FUNCTION_BLOCK FB_ManualMotionControl
VAR_INPUT
	
END_VAR
VAR_OUTPUT
END_VAR
VAR_IN_OUT
	stServoInterface		: stServoInterface;
END_VAR
VAR
	
	servoPower				: MC_Power;
	servoBuffer				: MC_BufferMode := MC_Aborting;
	
	servoReset				: MC_Reset;
	servoHome				: MC_Home;
	
	servoStatus				: MC_ReadStatus;
	
	servoSetPosition		: MC_SetPosition;
	
	servoJog				: MC_Jog;
	
	servoStop				: MC_Stop;
	
	servoMoveAbsolute		: MC_MoveAbsolute;
	
	servoMoveRelative		: MC_MoveRelative;
	
	servoMoveVelocity		: MC_MoveVelocity;
	
	jogErrorID				: UDINT;
	
	errorStop: BOOL;
	disabled: BOOL;
	stopping: BOOL;
	discreteMotion: BOOL;
	continuousMotion: BOOL;
	syncMotion: BOOL;
	homing: BOOL;
	constVelocity: BOOL;
	accel: BOOL;
	decel: BOOL;
	status: ST_AxisStatus;
	
	powerInterface 		: mcInterface;
	resetInterface		: mcInterface;
	homeInterface		: mcInterface;
	jogInterface		: mcInterface;
	stopInterface		: mcInterface;
	moveAbsInterface	: mcInterface;
	moveRelInterface	: mcInterface;
	moveVelInterface	: mcInterface;
	statusInterface		: mcInterface;
	
	// State Machine Variables
	startCycle			: BOOL;
	continueToTop		: BOOL;
	continueToBottom	: BOOL;
	endAtTop			: BOOL;
	endAtBottom			: BOOL;
	moveBottomTrig			: BOOL;
	moveTopTrig				: BOOL;
	
	demoState			: FB_ManualStateMachine;
	demoModePermissive	: BOOL;
	demoModeRun			: BOOL;
	bottomComplete		: BOOL;
	topComplete			: BOOL;
	
	servoMoveBottom		: MC_MoveAbsolute;
	servoMoveTop		: MC_MoveAbsolute;
	servoEstop			: MC_Halt;
	
	demoModePermissivesdf: INT;
END_VAR

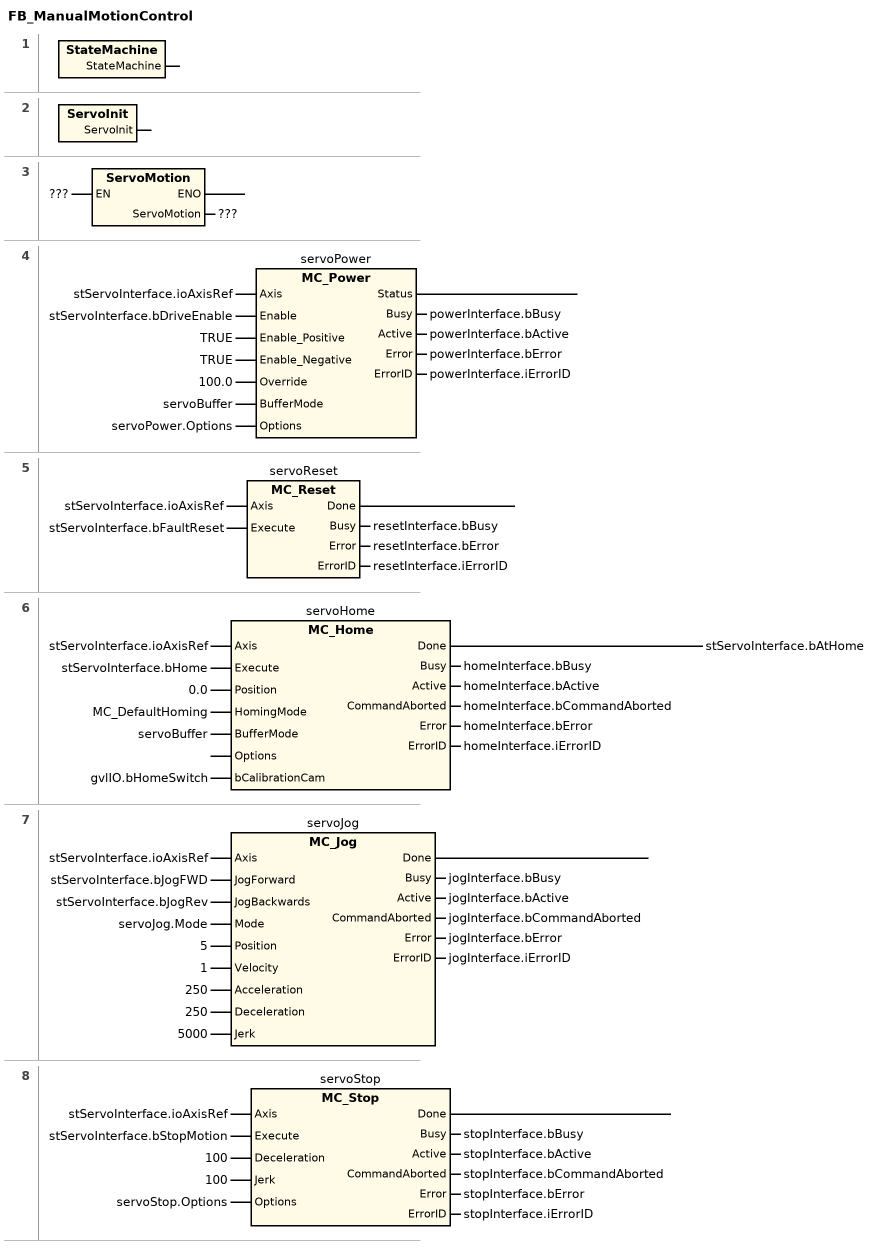
// NETWORK 1
StateMachine();

// NETWORK 2
ServoInit();

// NETWORK 3
ServoMotion();

// NETWORK 4
servoPower(
    Axis := stServoInterface.ioAxisRef,
    Enable := stServoInterface.bDriveEnable,
    Enable_Positive := TRUE,
    Enable_Negative := TRUE,
    Override := 100.0,
    BufferMode := servoBuffer,
    Options := servoPower.Options,
    Busy => powerInterface.bBusy,
    Active => powerInterface.bActive,
    Error => powerInterface.bError,
    ErrorID => powerInterface.iErrorID); // MC_Power

// NETWORK 5
servoReset(
    Axis := stServoInterface.ioAxisRef,
    Execute := stServoInterface.bFaultReset,
    Busy => resetInterface.bBusy,
    Error => resetInterface.bError,
    ErrorID => resetInterface.iErrorID); // MC_Reset

// NETWORK 6
servoHome(
    Axis := stServoInterface.ioAxisRef,
    Execute := stServoInterface.bHome,
    Position := 0.0,
    HomingMode := MC_DefaultHoming,
    BufferMode := servoBuffer,
    bCalibrationCam := gvlIO.bHomeSwitch,
    Busy => homeInterface.bBusy,
    Active => homeInterface.bActive,
    CommandAborted => homeInterface.bCommandAborted,
    Error => homeInterface.bError,
    ErrorID => homeInterface.iErrorID); // MC_Home
stServoInterface.bAtHome := servoHome.Done;

// NETWORK 7
servoJog(
    Axis := stServoInterface.ioAxisRef,
    JogForward := stServoInterface.bJogFWD,
    JogBackwards := stServoInterface.bJogRev,
    Mode := servoJog.Mode,
    Position := 5,
    Velocity := 1,
    Acceleration := 250,
    Deceleration := 250,
    Jerk := 5000,
    Busy => jogInterface.bBusy,
    Active => jogInterface.bActive,
    CommandAborted => jogInterface.bCommandAborted,
    Error => jogInterface.bError,
    ErrorID => jogInterface.iErrorID); // MC_Jog

// NETWORK 8
servoStop(
    Axis := stServoInterface.ioAxisRef,
    Execute := stServoInterface.bStopMotion,
    Deceleration := 100,
    Jerk := 100,
    Options := servoStop.Options,
    Busy => stopInterface.bBusy,
    Active => stopInterface.bActive,
    CommandAborted => stopInterface.bCommandAborted,
    Error => stopInterface.bError,
    ErrorID => stopInterface.iErrorID); // MC_Stop

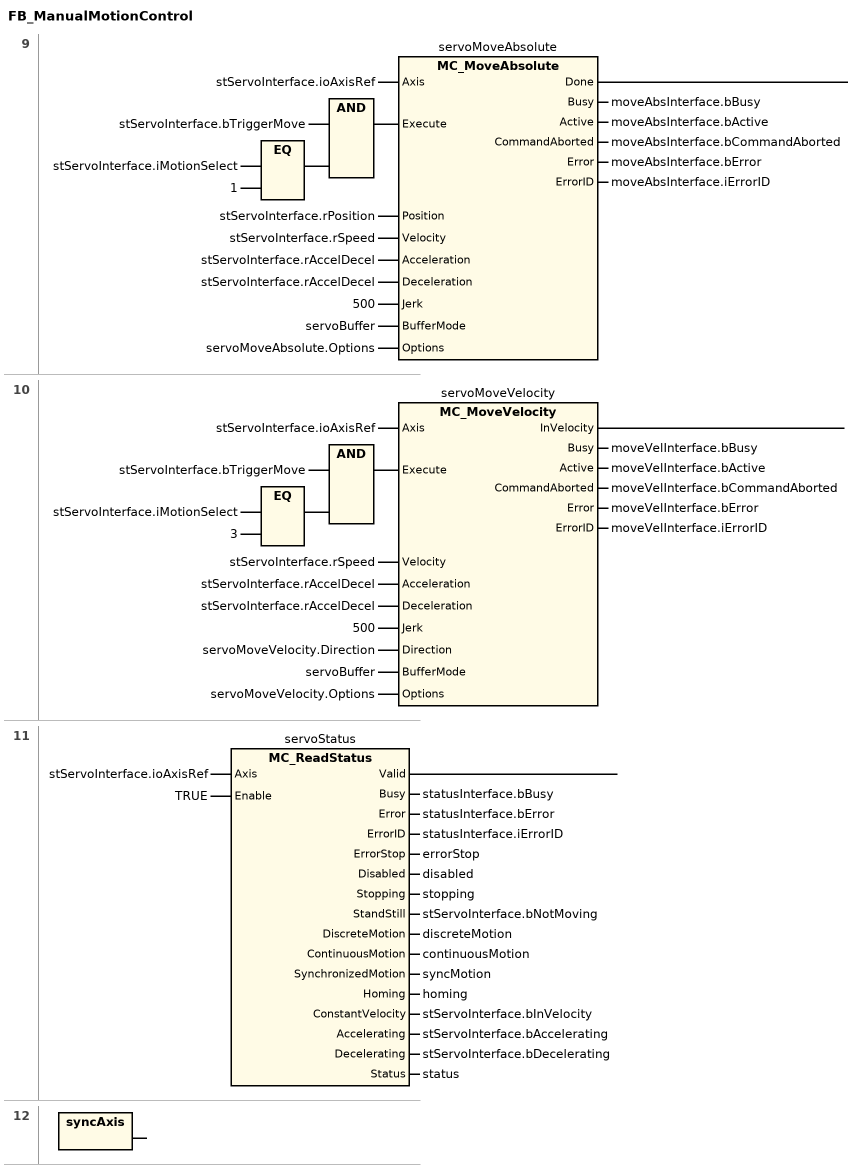
// NETWORK 9
servoMoveAbsolute(
    Axis := stServoInterface.ioAxisRef,
    Execute := stServoInterface.bTriggerMove AND stServoInterface.iMotionSelect = 1,
    Position := stServoInterface.rPosition,
    Velocity := stServoInterface.rSpeed,
    Acceleration := stServoInterface.rAccelDecel,
    Deceleration := stServoInterface.rAccelDecel,
    Jerk := 500,
    BufferMode := servoBuffer,
    Options := servoMoveAbsolute.Options,
    Busy => moveAbsInterface.bBusy,
    Active => moveAbsInterface.bActive,
    CommandAborted => moveAbsInterface.bCommandAborted,
    Error => moveAbsInterface.bError,
    ErrorID => moveAbsInterface.iErrorID); // MC_MoveAbsolute

// NETWORK 10
servoMoveVelocity(
    Axis := stServoInterface.ioAxisRef,
    Execute := stServoInterface.bTriggerMove AND stServoInterface.iMotionSelect = 3,
    Velocity := stServoInterface.rSpeed,
    Acceleration := stServoInterface.rAccelDecel,
    Deceleration := stServoInterface.rAccelDecel,
    Jerk := 500,
    Direction := servoMoveVelocity.Direction,
    BufferMode := servoBuffer,
    Options := servoMoveVelocity.Options,
    Busy => moveVelInterface.bBusy,
    Active => moveVelInterface.bActive,
    CommandAborted => moveVelInterface.bCommandAborted,
    Error => moveVelInterface.bError,
    ErrorID => moveVelInterface.iErrorID); // MC_MoveVelocity

// NETWORK 11
servoStatus(
    Axis := stServoInterface.ioAxisRef,
    Enable := TRUE,
    Busy => statusInterface.bBusy,
    Error => statusInterface.bError,
    ErrorID => statusInterface.iErrorID,
    ErrorStop => errorStop,
    Disabled => disabled,
    Stopping => stopping,
    StandStill => stServoInterface.bNotMoving,
    DiscreteMotion => discreteMotion,
    ContinuousMotion => continuousMotion,
    SynchronizedMotion => syncMotion,
    Homing => homing,
    ConstantVelocity => stServoInterface.bInVelocity,
    Accelerating => stServoInterface.bAccelerating,
    Decelerating => stServoInterface.bDecelerating,
    Status => status); // MC_ReadStatus

// NETWORK 12
syncAxis();

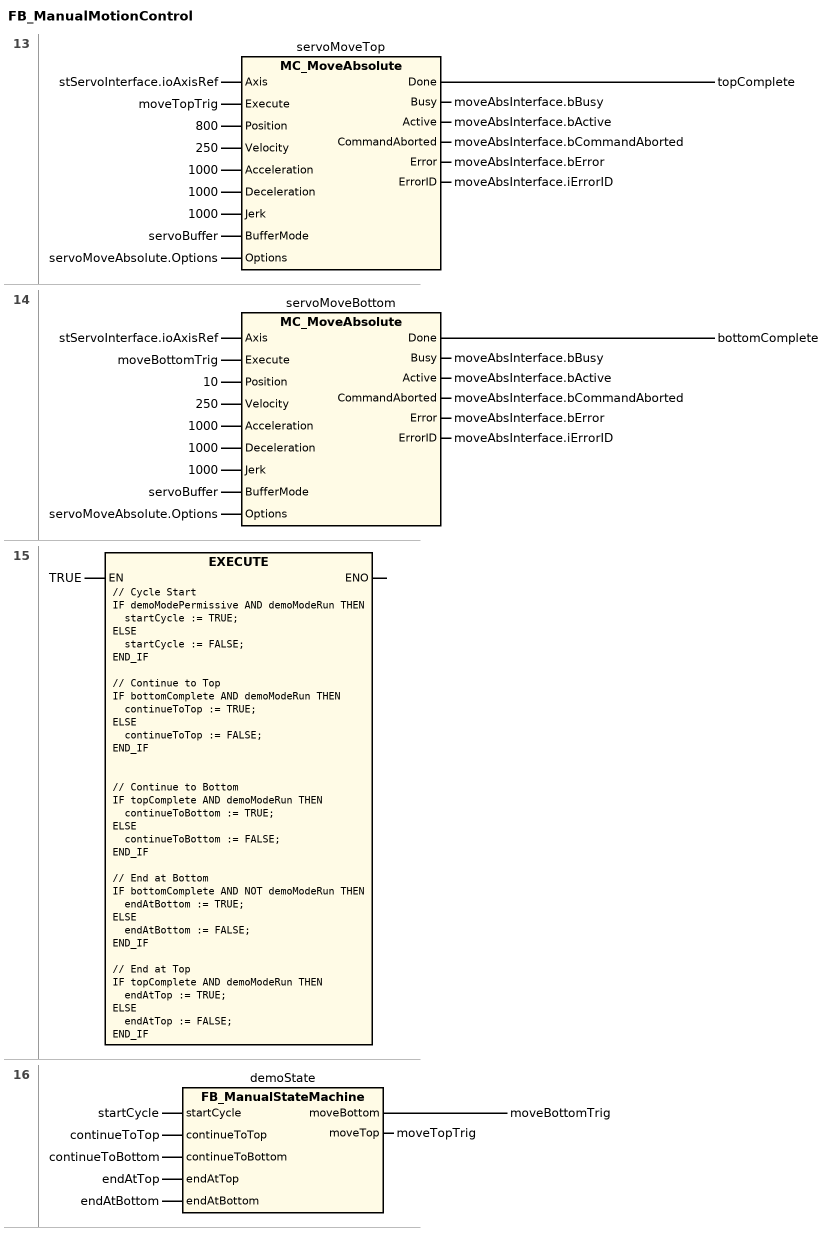
// NETWORK 13
servoMoveTop(
    Axis := stServoInterface.ioAxisRef,
    Execute := moveTopTrig,
    Position := 800,
    Velocity := 250,
    Acceleration := 1000,
    Deceleration := 1000,
    Jerk := 1000,
    BufferMode := servoBuffer,
    Options := servoMoveAbsolute.Options,
    Busy => moveAbsInterface.bBusy,
    Active => moveAbsInterface.bActive,
    CommandAborted => moveAbsInterface.bCommandAborted,
    Error => moveAbsInterface.bError,
    ErrorID => moveAbsInterface.iErrorID); // MC_MoveAbsolute
topComplete := servoMoveTop.Done;

// NETWORK 14
servoMoveBottom(
    Axis := stServoInterface.ioAxisRef,
    Execute := moveBottomTrig,
    Position := 10,
    Velocity := 250,
    Acceleration := 1000,
    Deceleration := 1000,
    Jerk := 1000,
    BufferMode := servoBuffer,
    Options := servoMoveAbsolute.Options,
    Busy => moveAbsInterface.bBusy,
    Active => moveAbsInterface.bActive,
    CommandAborted => moveAbsInterface.bCommandAborted,
    Error => moveAbsInterface.bError,
    ErrorID => moveAbsInterface.iErrorID); // MC_MoveAbsolute
bottomComplete := servoMoveBottom.Done;

// NETWORK 15
// Cycle Start
IF demoModePermissive AND demoModeRun THEN
	startCycle := TRUE;
ELSE 
	startCycle := FALSE;
END_IF

// Continue to Top
IF bottomComplete AND demoModeRun THEN
	continueToTop := TRUE;
ELSE
	continueToTop := FALSE;
END_IF


// Continue to Bottom
IF topComplete AND demoModeRun THEN
	continueToBottom := TRUE;
ELSE
	continueToBottom := FALSE;
END_IF

// End at Bottom
IF bottomComplete AND NOT demoModeRun THEN
	endAtBottom := TRUE;
ELSE
	endAtBottom := FALSE;
END_IF

// End at Top
IF topComplete AND demoModeRun THEN
	endAtTop := TRUE;
ELSE
	endAtTop := FALSE;
END_IF

// NETWORK 16
demoState(
    startCycle := startCycle,
    continueToTop := continueToTop,
    continueToBottom := continueToBottom,
    endAtTop := endAtTop,
    endAtBottom := endAtBottom,
    moveTop => moveTopTrig); // FB_ManualStateMachine
moveBottomTrig := demoState.moveBottom;

ACTION moveBottom:
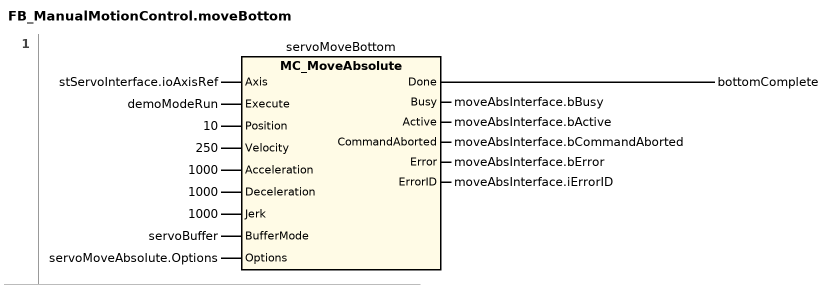
// NETWORK 1
servoMoveBottom(
    Axis := stServoInterface.ioAxisRef,
    Execute := demoModeRun,
    Position := 10,
    Velocity := 250,
    Acceleration := 1000,
    Deceleration := 1000,
    Jerk := 1000,
    BufferMode := servoBuffer,
    Options := servoMoveAbsolute.Options,
    Busy => moveAbsInterface.bBusy,
    Active => moveAbsInterface.bActive,
    CommandAborted => moveAbsInterface.bCommandAborted,
    Error => moveAbsInterface.bError,
    ErrorID => moveAbsInterface.iErrorID); // MC_MoveAbsolute
bottomComplete := servoMoveBottom.Done;
END_ACTION

ACTION moveTop:
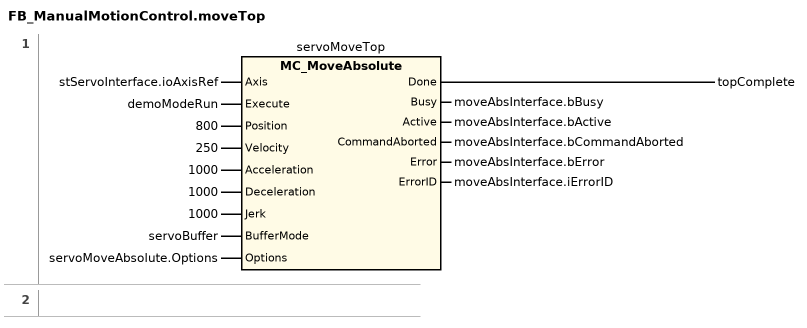
// NETWORK 1
servoMoveTop(
    Axis := stServoInterface.ioAxisRef,
    Execute := demoModeRun,
    Position := 800,
    Velocity := 250,
    Acceleration := 1000,
    Deceleration := 1000,
    Jerk := 1000,
    BufferMode := servoBuffer,
    Options := servoMoveAbsolute.Options,
    Busy => moveAbsInterface.bBusy,
    Active => moveAbsInterface.bActive,
    CommandAborted => moveAbsInterface.bCommandAborted,
    Error => moveAbsInterface.bError,
    ErrorID => moveAbsInterface.iErrorID); // MC_MoveAbsolute
topComplete := servoMoveTop.Done;

// NETWORK 2
END_ACTION

METHOD ServoInit : BOOL
VAR_INPUT
END_VAR
END_METHOD

METHOD ServoMotion : BOOL
VAR_INPUT
END_VAR
END_METHOD

METHOD StateMachine : BOOL
VAR_INPUT
END_VAR
END_METHOD

ACTION syncAxis:
CASE stServoInterface.ioAxisRef.NcToPlc.AxisState OF
	0 : // Inactive
	
	1 : // Running
		
	3 : // Phase_VeloConst
		stServoInterface.bInVelocity := TRUE;
	4 : // Phase_AccPos
		stServoInterface.bAccelerating := TRUE;
	5 : // Phase_AccNeg
		stServoInterface.bDecelerating := TRUE;
END_CASE

// Feedback

stServoInterface.rActualPosition := stServoInterface.ioAxisRef.NcToPlc.ActPos;

stServoInterface.rActualSpeed := stServoInterface.ioAxisRef.NcToPlc.ActVelo;

// Motion Status
stServoInterface.bDriveEnabled:= NOT(disabled);
stServoInterface.bMoving := NOT(stServoInterface.bNotMoving AND disabled);
stServoInterface.bFaulted := statusInterface.bError;

// Drive Control

// Demo Mode
IF stServoInterface.iMotionSelect = 1 THEN
	demoModePermissive := TRUE;
ELSE
	demoModePermissive := FALSE;
END_IF

IF demoModePermissive AND (stServoInterface.bDemoModeStart OR demoModeRun) AND NOT stServoInterface.bDemoModeStop THEN
	demoModeRun := TRUE;
ELSE
	demoModeRun := FALSE;
END_IF
END_ACTION

END_FUNCTION_BLOCK

(* stored: Version 1.1.0.1, ProductVersion 3.1.4024.12
   POU FB_ManualMotionControl: Id {6ef56c13-35f3-47e8-a8b0-04d3c6c54ada}, SpecialFunc None
   Action moveBottom: Id {11cd8f46-c3c7-4087-be07-77bc560d9d39}
   Action moveTop: Id {f11d386d-6a8a-47e5-ad35-164c0b176f2d}
   Method ServoInit: Id {0ce3093f-d820-433c-860b-d979707e5791}
   Method ServoMotion: Id {a34ff9e2-f41e-46ec-a835-e7a7cb60ec05}
   Method StateMachine: Id {2f8dffc0-6f8a-4476-9e0d-6463e510b9ea}
   Action syncAxis: Id {de180c65-aa7e-485b-a509-efecb712f169} *)
